# EPICS StreamDevice protocol: alexioc/test.proto
# streamDevice protocol file for general testing
#
#  $Revision: $
#  $Date: $
#  $Id: $
#  $Log: $
#
Terminator = CR;
ExtraInput = Ignore;
LockTimeout  = 2000;
ReplyTimeout = 300;
ReadTimeout  = 150;

CMDOUT {
	OUT "%s";
	#IN "%(DESC)s";
}

CMDIN {
	IN "%(ALEX:RDBYTE.A)3X";
}
